(* IEC 61131-3 sources: Industry-PLC-LLM/data/PLCBEAD_repo/PLCBEAD_PLCEmbed-main/PLC-BEAD/Source/GEB/_DWORD_TO_REAL, 1 file *)

(* ---- _DWORD_TO_REAL.ST ---- *)
FUNCTION _DWORD_TO_REAL:REAL
	VAR_INPUT
		IN :	DWORD;
	END_VAR

	_DWORD_TO_REAL := UDINT_TO_REAL(DWORD_TO_UDINT(IN));
END_FUNCTION

PROGRAM program0
  VAR
    LocalVar0 : DWORD;
    LocalOUT  : REAL;
  END_VAR

  LocalOUT := _DWORD_TO_REAL(LocalVar0);
END_PROGRAM
